// LS Electric XG5000 project: 32.Module 1~4 제어
// PLC NewPLC
// module base 0 slot 0: 입출력 모듈:XBM-DN/DP32HP (DC 24V입력/TR 출력, 32점)
// module base 0 slot 2: 입력 모듈:XBE-DC08A (DC 24V 입력, 8점 (전류소스 싱크공용))

PROGRAM NewProgram (task: 스캔 프로그램)

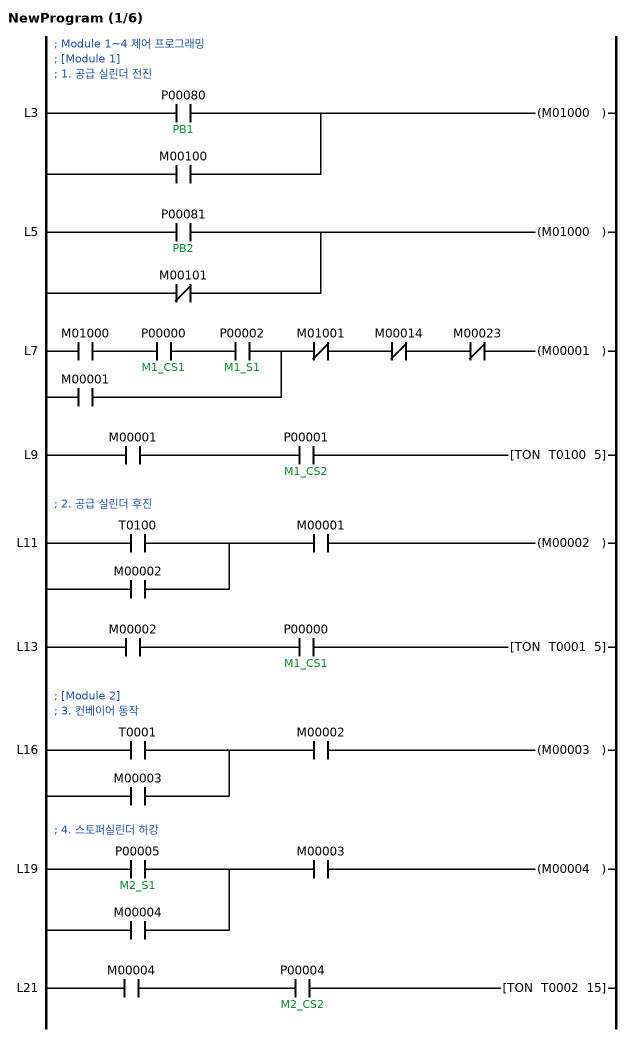
// Module 1~4 제어 프로그래밍
//  [Module 1]
// 1. 공급 실린더 전진
; L3
LOAD      P00080	// PB1
OR        M00100
OUT       M01000
; L5
LOAD      P00081	// PB2
OR NOT    M00101
OUT       M01000
; L7
LOAD      M01000
AND       P00000	// M1_CS1
AND       P00002	// M1_S1
OR        M00001
AND NOT   M01001
AND NOT   M00014
AND NOT   M00023
OUT       M00001
; L9
LOAD      M00001
AND       P00001	// M1_CS2
TON       T0100 5
// 2. 공급 실린더 후진
; L11
LOAD      T0100
OR        M00002
AND       M00001
OUT       M00002
; L13
LOAD      M00002
AND       P00000	// M1_CS1
TON       T0001 5
//  [Module 2]
// 3. 컨베이어 동작
; L16
LOAD      T0001
OR        M00003
AND       M00002
OUT       M00003
// 4. 스토퍼실린더 하강
; L19
LOAD      P00005	// M2_S1
OR        M00004
AND       M00003
OUT       M00004
; L21
LOAD      M00004
AND       P00004	// M2_CS2
TON       T0002 15

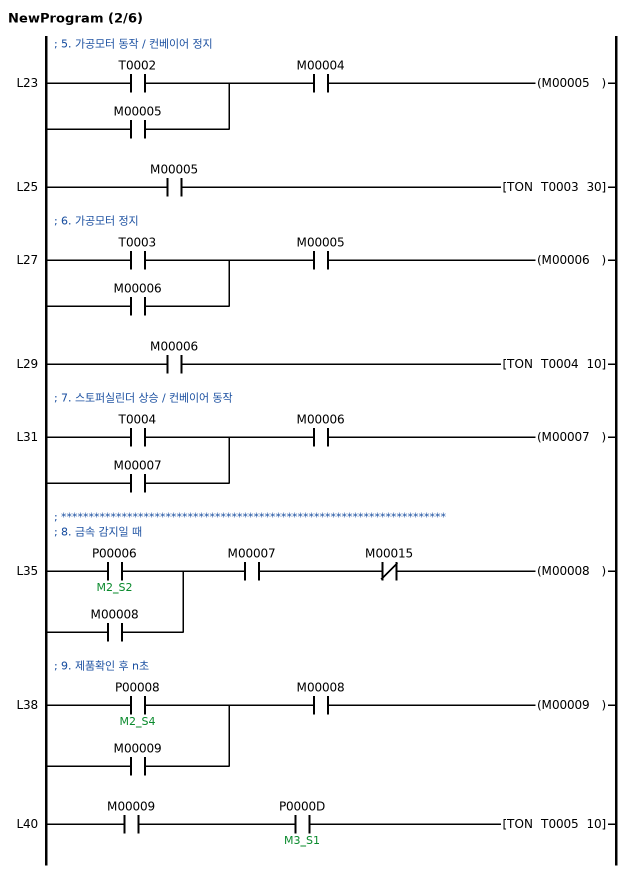
// 5. 가공모터 동작 / 컨베이어 정지
; L23
LOAD      T0002
OR        M00005
AND       M00004
OUT       M00005
; L25
LOAD      M00005
TON       T0003 30
// 6. 가공모터 정지
; L27
LOAD      T0003
OR        M00006
AND       M00005
OUT       M00006
; L29
LOAD      M00006
TON       T0004 10
// 7. 스토퍼실린더 상승 / 컨베이어 동작
; L31
LOAD      T0004
OR        M00007
AND       M00006
OUT       M00007
// **********************************************************************
// 8. 금속 감지일 때
; L35
LOAD      P00006	// M2_S2
OR        M00008
AND       M00007
AND NOT   M00015
OUT       M00008
// 9. 제품확인 후 n초
; L38
LOAD      P00008	// M2_S4
OR        M00009
AND       M00008
OUT       M00009
; L40
LOAD      M00009
AND       P0000D	// M3_S1
TON       T0005 10

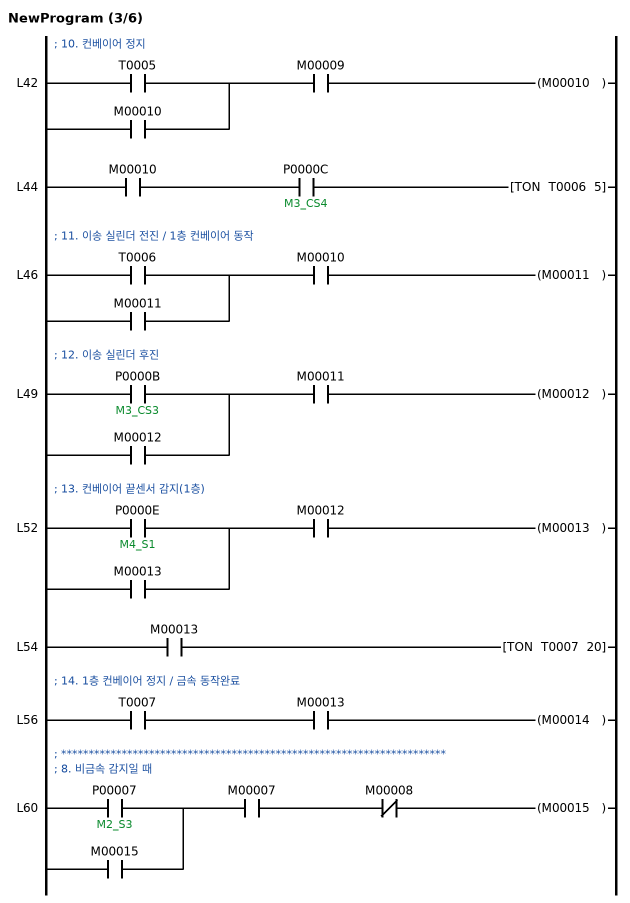
// 10. 컨베이어 정지
; L42
LOAD      T0005
OR        M00010
AND       M00009
OUT       M00010
; L44
LOAD      M00010
AND       P0000C	// M3_CS4
TON       T0006 5
// 11. 이송 실린더 전진 / 1층 컨베이어 동작
; L46
LOAD      T0006
OR        M00011
AND       M00010
OUT       M00011
// 12. 이송 실린더 후진
; L49
LOAD      P0000B	// M3_CS3
OR        M00012
AND       M00011
OUT       M00012
// 13. 컨베이어 끝센서 감지(1층)
; L52
LOAD      P0000E	// M4_S1
OR        M00013
AND       M00012
OUT       M00013
; L54
LOAD      M00013
TON       T0007 20
// 14. 1층 컨베이어 정지 / 금속 동작완료
; L56
LOAD      T0007
AND       M00013
OUT       M00014
// **********************************************************************
// 8. 비금속 감지일 때
; L60
LOAD      P00007	// M2_S3
OR        M00015
AND       M00007
AND NOT   M00008
OUT       M00015

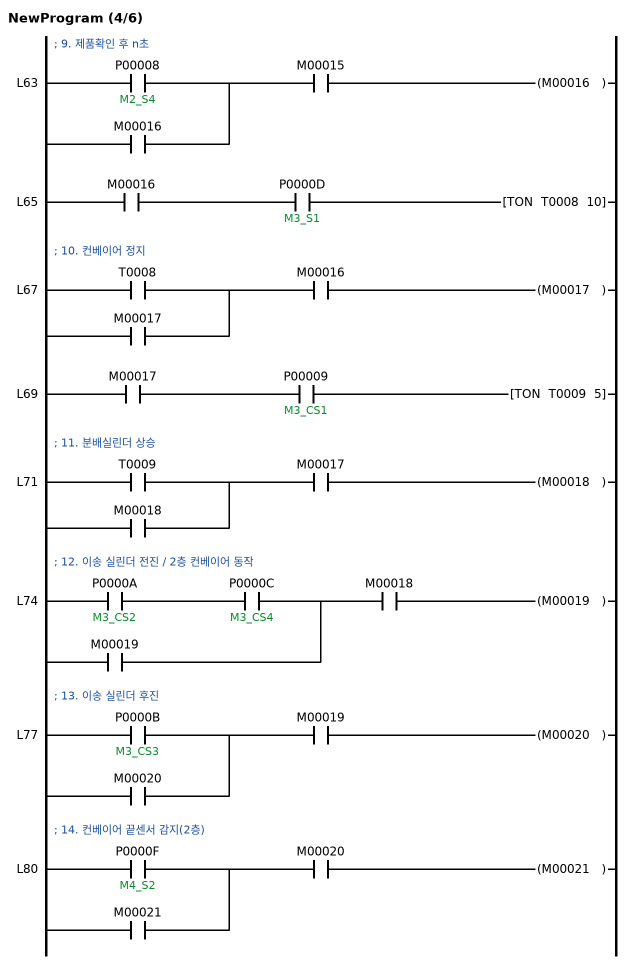
// 9. 제품확인 후 n초
; L63
LOAD      P00008	// M2_S4
OR        M00016
AND       M00015
OUT       M00016
; L65
LOAD      M00016
AND       P0000D	// M3_S1
TON       T0008 10
// 10. 컨베이어 정지
; L67
LOAD      T0008
OR        M00017
AND       M00016
OUT       M00017
; L69
LOAD      M00017
AND       P00009	// M3_CS1
TON       T0009 5
// 11. 분배실린더 상승
; L71
LOAD      T0009
OR        M00018
AND       M00017
OUT       M00018
// 12. 이송 실린더 전진 / 2층 컨베이어 동작
; L74
LOAD      P0000A	// M3_CS2
AND       P0000C	// M3_CS4
OR        M00019
AND       M00018
OUT       M00019
// 13. 이송 실린더 후진
; L77
LOAD      P0000B	// M3_CS3
OR        M00020
AND       M00019
OUT       M00020
// 14. 컨베이어 끝센서 감지(2층)
; L80
LOAD      P0000F	// M4_S2
OR        M00021
AND       M00020
OUT       M00021

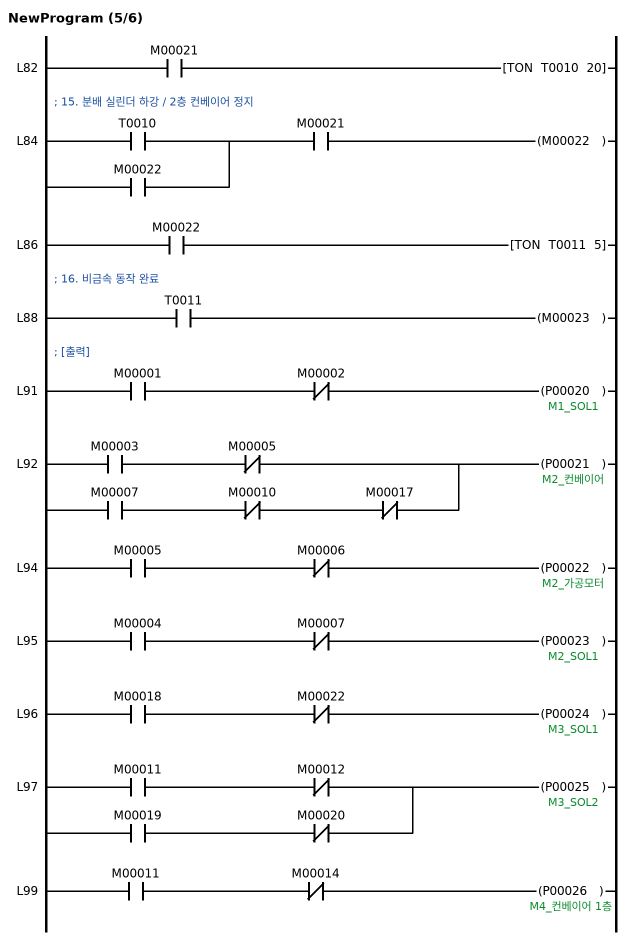
; L82
LOAD      M00021
TON       T0010 20
// 15. 분배 실린더 하강 / 2층 컨베이어 정지
; L84
LOAD      T0010
OR        M00022
AND       M00021
OUT       M00022
; L86
LOAD      M00022
TON       T0011 5
// 16. 비금속 동작 완료
; L88
LOAD      T0011
OUT       M00023
//  [출력]
; L91
LOAD      M00001
AND NOT   M00002
OUT       P00020	// M1_SOL1
; L92
LOAD      M00003
AND NOT   M00005
LOAD      M00007
AND NOT   M00010
AND NOT   M00017
OR LOAD
OUT       P00021	// M2_컨베이어
; L94
LOAD      M00005
AND NOT   M00006
OUT       P00022	// M2_가공모터
; L95
LOAD      M00004
AND NOT   M00007
OUT       P00023	// M2_SOL1
; L96
LOAD      M00018
AND NOT   M00022
OUT       P00024	// M3_SOL1
; L97
LOAD      M00011
AND NOT   M00012
LOAD      M00019
AND NOT   M00020
OR LOAD
OUT       P00025	// M3_SOL2
; L99
LOAD      M00011
AND NOT   M00014
OUT       P00026	// M4_컨베이어 1층

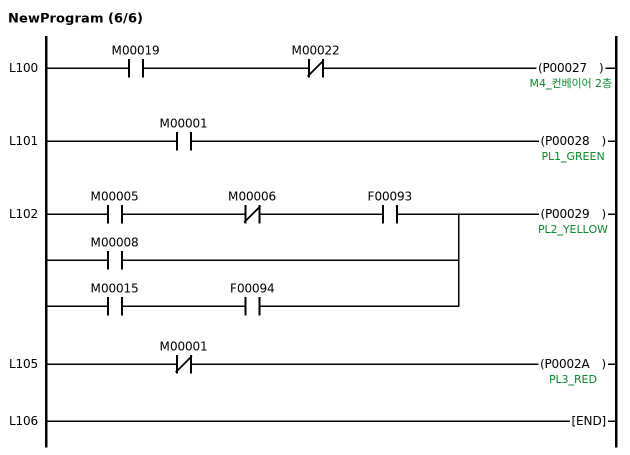
; L100
LOAD      M00019
AND NOT   M00022
OUT       P00027	// M4_컨베이어 2층
; L101
LOAD      M00001
OUT       P00028	// PL1_GREEN
; L102
LOAD      M00005
AND NOT   M00006
AND       F00093
OR        M00008
LOAD      M00015
AND       F00094
OR LOAD
OUT       P00029	// PL2_YELLOW
; L105
LOAD NOT  M00001
OUT       P0002A	// PL3_RED
; L106
END

VARIABLES AND COMMENTS (devices not used above)
P00083	BIT	PB4
P00082	BIT	PB3
P00003	BIT	M2_CS1